TYPE "LBP_typeHMI"
TITLE = Operator panel signals / Signaux pupitre opérateur
// User data type for block LBP_HMI [DB19] / Type de données utilisateur pour bloc LBP_HMI [DB19]
   STRUCT
      A_SCLight : Bool;   // Screen light / Éclaircir écran
      A_SCDark : Bool;   // Screen darkening / Obscurcissement écran
      A_KeyDisable : Bool;   // Key disable / Désactiver touche
      A_ClearCanAl : Bool;   // Clear cancel alarms / Supprimer alarmes d'abandon
      A_ClearRecAl : Bool;   // Clear recall alarms / Supprimer alarmes de rappel
      f0_5 : Bool;
      A_SafeActionLog : Bool;   // Edge change 0 → 1: Save ACTION.COM to CRASH.COM / Front 0 → 1 : enregistrer ACTION.COM dans CRASH.COM
      A_ActWCS : Bool;   // Actual value in WCS 0=MCS / Valeur réelle dans WCS 0=MCS
      A_PLCExtViewerReject : Bool;   // External viewer reject / Refuser visualiseur externe
      A_PLCExtViewerMode : Bool;   // External viewer mode / Mode visualiseur externe
      f1_2 : Bool;
      f1_3 : Bool;
      f1_4 : Bool;
      f1_5 : Bool;
      f1_6 : Bool;
      f1_7 : Bool;
      A_1stError1 : Word;   // 1st error HIGRAPH / 1re erreur HIGRAPH
      A_1stError2 : Word;   // 1st error HIGRAPH / 1re erreur HIGRAPH
      A_ASpi1percent : Byte;   // Analog spindle 1: / Broche analogique 1 :
      A_ASpi2percent : Byte;
      A_MCPChan : Byte;
      A_OEM1 : Bool;
      A_OEM2 : Bool;
      A_AToolMeas : Bool;   // AutoToolMeasure
      f9_3 : Bool;
      f9_4 : Bool;
      f9_5 : Bool;
      f9_6 : Bool;
      f9_7 : Bool;
      A_Hardkey : Byte;   // PLC hardkeys / Touches matérielles AP
      f11 : Byte;   // Reserved for hardkeys / Réservé pour touches matérielles
      f12_0 : Bool;
      f12_1 : Bool;
      A_COM2 : Bool;
      A_COM1 : Bool;
      A_V24stop : Bool;
      A_V24ext : Bool;
      A_V24off : Bool;
      A_V24on : Bool;
      A_TeachDisable : Bool;
      f13_1 : Bool;
      f13_2 : Bool;
      f13_3 : Bool;
      f13_4 : Bool;
      A_PPdeload : Bool;
      A_PPload : Bool;
      A_PPsel : Bool;
      A_V24Index1 : Byte;
      A_V24Index2 : Byte;
      A_V24NoFile1 : Byte;
      A_V24NoFile2 : Byte;
      A_res18 : Byte;
      A_res19 : Byte;   // Message counter / Compteur de messages
      f20_0 : Bool;
      E_SCDark : Bool;   // Screen darkening / Obscurcissement écran
      E_Cancel : Bool;   // Cancel / Abandon
      E_CanCleared : Bool;   // Cancel alarms cleared / Alarmes d'abandon supprimées
      E_RecCleared : Bool;   // Recall alarms cleared / Alarmes de rappel supprimées
      f20_5 : Bool;   // res. language / rés. langue
      E_SimActiv : Bool;   // Simulation active
      E_ActWCS : Bool;   // Switchover MCS/WCS 0=MCS / Commutation MCS/WCS 0=MCS
      E_ActivWA : Byte;
      E_Chan : Byte;   // Channel displayed / Canal affiché
      E_KeybHandl : Bool;   // Keyboard handling / Gestion clavier
      E_DataTransf : Bool;   // Data transfer active / Transmission de données active
      E_DisplChange : Bool;   // Display change / Modification affichage
      f23_3 : Bool;
      f23_4 : Bool;
      f23_5 : Bool;
      f23_6 : Bool;
      f23_7 : Bool;
      E_ScreenNo : Word;
      E_res26_0 : Bool;   // Reserved / Réservé
      E_PPOK : Bool;   // Part program status OK / État programme pièce OK
      E_PPErr : Bool;   // Part program status error / Programme pièce erreur d'état
      E_PPAct : Bool;   // Part program status active / État programme pièce actif
      f26_4 : Bool;   // Reserved / Réservé
      E_PPdeload : Bool;   // Part program status deloading / État programme pièce en cours de déchargement
      E_PPload : Bool;   // Part program status loading / État programme pièce en cours de chargement
      E_PPsel : Bool;   // Part program status selecting / État programme pièce en cours de sélection
      E_PPError : Byte;   // Part program status error / Programme pièce erreur d'état
      A_PictNo : Int;
      A_PictOn : Bool;
      A_PictOff : Bool;
      f30_2 : Bool;
      f30_3 : Bool;
      f30_4 : Bool;
      f30_5 : Bool;
      f30_6 : Bool;
      f30_7 : Bool;
      E_PictOK : Bool;
      E_PictOn : Bool;
      E_PictAct : Bool;
      E_PictOff : Bool;
      E_PictErr : Bool;
      f31_5 : Bool;
      f31_6 : Bool;
      E_NotAct : Bool;
      A_FuncNo : Byte;
      A_Par1 : Byte;
      A_Par2 : Byte;
      A_Par3 : Byte;
      E_FuncErr : Byte;
      f37 : Byte;
      f38 : Byte;
      f39 : Byte;
      res40 : Array[0..9] of Byte;
      MMC2 : Struct
         A_SCLight : Bool;   // Screen light / Éclaircir écran
         A_SCDark : Bool;   // Screen darkening / Obscurcissement écran
         A_KeyDisable : Bool;   // Key disable / Désactiver touche
         A_ClearCanAl : Bool;   // Clear cancel alarms / Supprimer alarmes d'abandon
         A_ClearRecAl : Bool;   // Clear recall alarms / Supprimer alarmes de rappel
         f0_5 : Bool;
         f0_6 : Bool;
         A_ActWCS : Bool;   // Actual value in WCS 0=MCS / Valeur réelle dans WCS 0=MCS
         A_PLCExtViewerReject : Bool;   // External viewer reject / Refuser visualiseur externe
         A_PLCExtViewerMode : Bool;   // External viewer mode / Mode visualiseur externe
         f1_2 : Bool;
         f1_3 : Bool;
         f1_4 : Bool;
         f1_5 : Bool;
         f1_6 : Bool;
         f1_7 : Bool;
         A_1stError1 : Word;   // 1st error HIGRAPH / 1re erreur HIGRAPH
         A_1stError2 : Word;   // 1st error HIGRAPH / 1re erreur HIGRAPH
         A_ASpi1percent : Byte;   // Analog spindle 1: / Broche analogique 1 :
         A_ASpi2percent : Byte;
         A_MCPChan : Byte;
         A_OEM1 : Bool;
         A_OEM2 : Bool;
         A_AToolMeas : Bool;   // AutoToolMeasure
         f9_3 : Bool;
         f9_4 : Bool;
         f9_5 : Bool;
         f9_6 : Bool;
         f9_7 : Bool;
         A_Hardkey : Byte;   // PLC hardkeys / Touches matérielles AP
         f11 : Byte;   // Reserved for hardkeys / Réservé pour touches matérielles
         f12_0 : Bool;
         f12_1 : Bool;
         A_COM2 : Bool;
         A_COM1 : Bool;
         A_V24stop : Bool;
         A_V24ext : Bool;
         A_V24off : Bool;
         A_V24on : Bool;
         A_TeachDisable : Bool;
         f13_1 : Bool;
         f13_2 : Bool;
         f13_3 : Bool;
         f13_4 : Bool;
         A_PPdeload : Bool;
         A_PPload : Bool;
         A_PPsel : Bool;
         A_V24Index1 : Byte;
         A_V24Index2 : Byte;
         A_V24NoFile1 : Byte;
         A_V24NoFile2 : Byte;
         A_res18 : Byte;
         A_res19 : Byte;   // Message counter / Compteur de messages
         f20_0 : Bool;
         E_SCDark : Bool;   // Screen darkening / Obscurcissement écran
         E_Cancel : Bool;   // Cancel / Abandon
         E_CanCleared : Bool;   // Cancel alarms cleared / Alarmes d'abandon supprimées
         E_RecCleared : Bool;   // Recall alarms cleared / Alarmes de rappel supprimées
         f20_5 : Bool;   // res. language / rés. langue
         E_SimActiv : Bool;   // Simulation active
         E_ActWCS : Bool;   // Switchover MCS/WCS 0=MCS / Commutation MCS/WCS 0=MCS
         E_ActivWA : Byte;
         E_Chan : Byte;   // Channel displayed / Canal affiché
         E_KeybHandl : Bool;   // Keyboard handling / Gestion clavier
         E_DataTransf : Bool;   // Data transfer active / Transmission de données active
         E_DisplChange : Bool;   // Display change / Modification affichage
         f23_3 : Bool;
         f23_4 : Bool;
         f23_5 : Bool;
         f23_6 : Bool;
         f23_7 : Bool;
         E_ScreenNo : Word;
         E_res26_0 : Bool;   // Reserved / Réservé
         E_PPOK : Bool;   // Part program status OK / État programme pièce OK
         E_PPErr : Bool;   // Part program status error / Programme pièce erreur d'état
         E_PPAct : Bool;   // Part program status active / État programme pièce actif
         f26_4 : Bool;   // Reserved / Réservé
         E_PPdeload : Bool;   // Part program status deloading / État programme pièce en cours de déchargement
         E_PPload : Bool;   // Part program status loading / État programme pièce en cours de chargement
         E_PPsel : Bool;   // Part program status selecting / État programme pièce en cours de sélection
         E_PPError : Byte;   // Part program status error / Programme pièce erreur d'état
         A_PictNo : Int;
         A_PictOn : Bool;
         A_PictOff : Bool;
         f30_2 : Bool;
         f30_3 : Bool;
         f30_4 : Bool;
         f30_5 : Bool;
         f30_6 : Bool;
         f30_7 : Bool;
         E_PictOK : Bool;
         E_PictOn : Bool;
         E_PictAct : Bool;
         E_PictOff : Bool;
         E_PictErr : Bool;
         f31_5 : Bool;
         f31_6 : Bool;
         E_NotAct : Bool;
         A_FuncNo : Byte;
         A_Par1 : Byte;
         A_Par2 : Byte;
         A_Par3 : Byte;
         E_FuncErr : Byte;
         f37 : Byte;
         f38 : Byte;
         f39 : Byte;
         res40 : Array[0..9] of Byte;
      END_STRUCT;
      ONL_REQUEST : Word;
      ONL_CONFIRM : Word;
      PAR_CLIENT_IDENT : Word;
      PAR_MMC_TYP : Byte;
      PAR_MSTT_ADR : Byte;
      PAR_STATUS : Byte;
      PAR_Z_INFO : Byte;
      MtoNAlive : Word;
      f112 : Byte;
      ParOpKeyAdr : Byte;
      ParTcuIndex : Byte;
      f115 : Byte;
      Tcu1KeyAdr : Byte;
      Tcu2KeyAdr : Byte;
      Tcu1Index : Byte;
      Tcu2Index : Byte;
      MMC1_CLIENT_IDENT : Word;
      MMC1_TYP : Byte;
      MMC1_MSTT_ADR : Byte;
      MMC1_STATUS : Byte;
      MMC1_Z_INFO : Byte;
      MMC1_SHIFT_LOCK : Bool;
      MMC1_MSTT_SHIFT_LOCK : Bool;
      MMC1_ACTIVE_REQ : Bool;
      MMC1_ACTIVE_PERM : Bool;
      MMC1_ACTIVE_CHANGED : Bool;
      MMC1_CHANGED_DENIED : Bool;
      MMC1_TCU_SHIFT_LOCK : Bool;
      f127 : Byte;
      MMC1_TRANS_DB : Word;
      MMC2_CLIENT_IDENT : Word;
      MMC2_TYP : Byte;
      MMC2_MSTT_ADR : Byte;
      MMC2_STATUS : Byte;
      MMC2_Z_INFO : Byte;
      MMC2_SHIFT_LOCK : Bool;
      MMC2_MSTT_SHIFT_LOCK : Bool;
      MMC2_ACTIVE_REQ : Bool;
      MMC2_ACTIVE_PERM : Bool;
      MMC2_ACTIVE_CHANGED : Bool;
      MMC2_CHANGED_DENIED : Bool;
      MMC2_TCU_SHIFT_LOCK : Bool;
      f137 : Byte;
      MMC2_TRANS_DB : Word;
      A_Subtype : Int;   // For code carrier Input from PLC / Pour porte-code entrée par AP
      A_Duplo : Int;
      A_Ident : String[32];
      A_Tnumber : Int;
      A_MagazinePlace : Int;
      A_MagazinePlaceType : Int;
      A_ToolSize_Upper : Byte;
      A_ToolSize_Down : Byte;
      A_ToolSize_Left : Byte;
      A_ToolSize_Right : Byte;
      A_Channel : Byte;
      A_LoadingPlace : Byte;
      A_Magazine : Int;
      A_Unit : Byte;
      A_NCU_Index : Byte;
      A_FileIndex : Int;
      A_ActiveEnable : Bool;
      A_Override : Bool;
      A_LoadTool : Bool;
      A_DeleteTool : Bool;
      E_Subtype : Int;   // For code carrier Output to PLC / Pour porte-code sortie vers AP
      E_Duplo : Int;
      E_Ident : String[32];
      E_Tnumber : Int;
      E_ToolState : Int;
      E_MagazinePlaceType : Int;
      E_ToolSize_Upper : Byte;
      E_ToolSize_Down : Byte;
      E_ToolSize_Left : Byte;
      E_ToolSize_Right : Byte;
      E_Magazine : Int;
      E_MagazinePlace : Int;
      A_ReqMMC1 : Bool;   // For code carrier Request MMC-Interface1 / Pour porte-code demander interface MMC1
      A_ReqMMC2 : Bool;   // For code carrier Request MMC-Interface2 / Pour porte-code demander interface MMC2
      A_K_Code : Byte;
      E_Done : Bool;
      E_Error : Bool;
      E_Active : Bool;
      f252_3 : Bool;
      f252_4 : Bool;
      f252_5 : Bool;
      f252_6 : Bool;
      E_Ident_Ready : Bool;
      E_K_CodeError : Byte;   // Identify for Error_Code / Identifier pour Error_Code
      E_Error_Code : Int;
      E_Req : Bool;   // For Positioning / Pour positionnement
      f257 : Byte;
      A_Done : Bool;
      A_Error : Bool;
      A_Active : Bool;
      f258_3 : Bool;
      f258_4 : Bool;
      f258_5 : Bool;
      f258_6 : Bool;
      f258_7 : Bool;
      E_TDC_Read : Bool;
      E_TDC_Write : Bool;
      E_TDC_Cancel : Bool;
      E_TDC_Read_before_Write : Bool;
      f259_4 : Bool;
      f259_5 : Bool;
      f259_6 : Bool;
      f259_7 : Bool;
      A_Error_Code : Int;
      E_PMagazine : Int;
      E_PMagazinePlace : Int;
      E_PTnumber : Int;   // TPM data / Données TPM
      A_TPMStatus : Int;
      A_TPMCounter : Array[1..32] of DInt;
      A_HWeelSimOvr : Byte;
      f399 : Byte;
      A_SimOvr : Int;   // Simulation override / Correction simulation
      A_SimState : Int;   // Simulation state / État simulation
      E_HmiUserKey : Array[1..64] of Bool;   // HMI user keys for HMI sidescreen / HMI touches utilisateur pour écran latéral IHM
      A_HmiUserLed : Array[1..64] of Bool;   // LEDs to the user keys for HMI sidescreen / LED pour touches utilisateur pour écran latéral IHM
      A_DisableHmiUserKey : Array[1..64] of Bool;   // Disable user keys for HMI sidescreen / Désactiver les touches utilisateur pour écran latéral IHM
      SafetyAutoAcceptanceTest : Struct   // Interface for the automated acceptance test
         E_Prepare : Bool;   // Prepare automated acceptance test requested by client
         E_Finalize : Bool;   // Stop automated acceptance test requested by client
         E_Cancel : Bool;   // Cancel automated acceptance test requested by client
         E_Perform : Bool;   // Perform automated acceptance test requested by client
         E_PerformSequence : Bool;   // Perform entire test sequence for automated acceptance test requested by client
         f428_5 : Bool;
         f428_6 : Bool;
         f428_7 : Bool;
         f429 : Byte;
         A_Prepared : Bool;   // Automated acceptance test was successfully prepared
         A_Finalized : Bool;   // Automated acceptance test was successfully stopped
         A_Canceled : Bool;   // Automated acceptance test was canceled successfully
         A_Performed : Bool;   // Automated acceptance test was performed successfully
         A_SequencePerformed : Bool;   // Entire test sequence for automated acceptance test is running
         f430_5 : Bool;
         f430_6 : Bool;
         f430_7 : Bool;
         f431_0 : Bool;
         A_Error : Bool;   // Automated acceptance test was canceled
         A_InvalidGroup : Bool;   // Test group is not accepted
         A_InvalidNumber : Bool;   // Test number is not accepted
         f431_4 : Bool;
         f431_5 : Bool;
         f431_6 : Bool;
         f431_7 : Bool;
         E_Group : Int;   // Test group for the current test
         E_Number : Int;   // Test number for the current test
         E_AxisNumber : Int;   // Axis number for the current test
         E_TraversePlus : Bool;   // Traversing direction for the current test (FALSE=negative, TRUE=positive)
         E_SelectSafeStop : Bool;   // Safe Stop is set for the current test
         E_SelectBrake : Bool;   // Brake used for the current test. (FALSE=Brake1, TRUE=Brake2)
         E_SelectSbtMode : Bool;   // SBT Test Sequence used for the current test. (FALSE=Sequence1, TRUE=Sequence2)
         E_SelectSlpMode : Int;   // Safe End Position used for the current test. ("SE/SLP PositionArea" : 1=SE1 ; 2=SE2)
         E_SelectSlsMode : Int;   // Safe Speed (SG1..SG4) used for the current test
      END_STRUCT;
   END_STRUCT;
END_TYPE

TYPE "LBP_typeInternal1"
TITLE = Internal data type for basic program / Type de données interne pour programme de base
// Data type only for internal use in the basic program / Type de données réservé à l'utilisation interne dans le programme de base
   STRUCT
      active : Bool;
      mcpAddress : USInt;
      modeDCK : Bool;
      clientPort : UInt;
      connectionId : CONN_OUC;
      mcpClientReference : Word;
      mcpInPointer : Struct
         DbNumber : Word;
         PointerAddress : DWord;
      END_STRUCT;
      mcpOutPointer : Struct
         DbNumber : Word;
         PointerAddress : DWord;
      END_STRUCT;
      mcpDefaultInLength : UInt;
      mcpDefaultOutLength : UInt;
      useIpAddress : Bool;
      ipAddress : Array[1..4] of USInt;
   END_STRUCT;
END_TYPE

TYPE "LBP_typeInternal2"
TITLE = Internal data type for basic program / Type de données interne pour programme de base
// Data type only for internal use in the basic program / Type de données réservé à l'utilisation interne dans le programme de base
   STRUCT
      "Version" { ExternalAccessible := 'False'; ExternalVisible := 'False'; ExternalWritable := 'False'} : UDInt;
      ObNumber { ExternalAccessible := 'False'; ExternalVisible := 'False'; ExternalWritable := 'False'} : UDInt;
   END_STRUCT;
END_TYPE

TYPE "LBP_typeInternal3"
TITLE = Internal data type for basic program / Type de données interne pour programme de base
// Data type only for internal use in the basic program / Type de données réservé à l'utilisation interne dans le programme de base
   STRUCT
      "Version" { ExternalAccessible := 'False'; ExternalVisible := 'False'; ExternalWritable := 'False'} : UDInt;
      BlockReturnValue { ExternalAccessible := 'False'; ExternalVisible := 'False'; ExternalWritable := 'False'} : UDInt;
      AlarmList { ExternalAccessible := 'False'; ExternalVisible := 'False'; ExternalWritable := 'False'} : Array[1..6] of Struct
         ARID : UInt;
         AlarmMessage : Bool;
         OperationMessage : Bool;
         AlarmIsComing : Bool;
         StopPlc : Bool;
         NumberOfExtendedValues : USInt;
         AlarmNumber : UDInt;
         ExtendedValueList : Array[1..9] of UDInt;
      END_STRUCT;
   END_STRUCT;
END_TYPE

TYPE "LBP_typeInternal4"
TITLE = Internal data type for basic program / Type de données interne pour programme de base
// Data type only for internal use in the basic program / Type de données réservé à l'utilisation interne dans le programme de base
   STRUCT
      Handwheels : Array[1..6] of Struct
         active : Bool;
         recent : Bool;
         stopped : Bool;
         pulses : Int;
      END_STRUCT;
   END_STRUCT;
END_TYPE

TYPE "LBP_typeInternal5"
TITLE = Internal data type for basic program / Type de données interne pour programme de base
// Data type only for internal use in the basic program / Type de données réservé à l'utilisation interne dans le programme de base
   STRUCT
      accepted : Bool;
      abort : Bool;
      writeRecord : Bool;
      mcpNumber : UInt;
      slotNumber : UInt;
      recordNumber : UInt;
      recordLength : UInt;
      recordData : Array[0..223] of Byte;
      done : Bool;
      busy : Bool;
      error : Bool;
      status : Word;
   END_STRUCT;
END_TYPE

TYPE "LBP_typeModeGroup"
TITLE = Mode group signals / Signaux groupe de modes de fonctionnement
// User data type for block LBP_ModeGroup [DB11] / Type de données utilisateur pour bloc LBP_ModeGroup [DB11]
   STRUCT
      A_AUTO : Bool;   // Operating mode AUTOMATIC / Mode AUTOMATIC
      A_MDA : Bool;   // Operating mode MDA / Mode MDA
      A_JOG : Bool;   // Operating mode JOG / Mode JOG
      f0_3 : Bool;
      A_MCDisable : Bool;   // Mode change disable / Désactiver changement mode de fonctionnement
      A_MGStop : Bool;   // Mode group stop / Groupe de modes de fonctionnement Arrêt
      A_MGStopASp : Bool;   // Mode group stop axes plus spindle / Groupe de modes de fonctionnement Arrêt axes et broche
      A_MGReset : Bool;   // Mode group reset / Groupe de modes de fonctionnement Reset
      A_TEACHIN : Bool;   // Machine function TEACH IN / Fonction machine TEACH IN
      A_REPOS : Bool;   // Machine function REPOS / Fonction machine REPOS
      A_REF : Bool;   // Machine function REF / Fonction machine REF
      f1_3 : Bool;
      f1_4 : Bool;
      f1_5 : Bool;
      A_SingleBlock_B : Bool;   // Single block type B / Bloc par bloc type B
      A_SingleBlock_A : Bool;   // Single block type A / Bloc par bloc type A
      A_INC1 : Bool;   // INC1
      A_INC10 : Bool;   // INC10
      A_INC100 : Bool;   // INC100
      A_INC1000 : Bool;   // INC1000
      A_INC10000 : Bool;   // INC10000
      A_INCVar : Bool;   // INC variable / Variable INC
      A_ContManTravel : Bool;   // Continuous manual travel / Mode manuel continu
      f2_7 : Bool;
      f3 : Byte;
      E_MMC_AUTO : Bool;   // HMI mode strobe AUTOMATIC / HMI mode Strobe AUTOMATIC
      E_MMC_MDA : Bool;   // HMI mode strobe MDA / HMI mode Strobe MDA
      E_MMC_JOG : Bool;   // HMI mode strobe JOG / HMI mode Strobe JOG
      f4_3 : Bool;
      f4_4 : Bool;
      f4_5 : Bool;
      f4_6 : Bool;
      f4_7 : Bool;
      E_MMC_TEACHIN : Bool;   // HMI machine function strobe TEACH IN / HMI Fonction machine Strobe TEACH IN
      E_MMC_REPOS : Bool;   // HMI machine function strobe REPOS / HMI Fonction machine Strobe REPOS
      E_MMC_REF : Bool;   // HMI machine function strobe REF / HMI Fonction machine Strobe REF
      f5_3 : Bool;
      f5_4 : Bool;
      f5_5 : Bool;
      f5_6 : Bool;
      f5_7 : Bool;
      E_AUTO : Bool;   // Active operating mode AUTOMATIC / Mode actif AUTOMATIC
      E_MDA : Bool;   // Active operating mode MDA / Mode actif MDA
      E_JOG : Bool;   // Active operating mode JOG / Mode actif JOG
      E_MGOK : Bool;   // Mode group ready / Groupe de modes de fonctionnement prêt
      E_MGreseted : Bool;   // Mode group reset performed / Groupe de modes de fonctionnement Reset effectué
      E_NCKintJOG : Bool;   // NCK internal JOG active / NCK JOG interne actif
      f6_6 : Bool;
      E_ChanReset : Bool;   // All channels in reset state / Tous les canaux en mode Reset
      E_TEACHIN : Bool;   // Active machine function TEACH IN / Fonction machine active TEACH IN
      E_REPOS : Bool;   // Active machine function REPOS / Fonction machine active REPOS
      E_REF : Bool;   // Active machine function REF / Fonction machine active REF
      f7_3 : Bool;
      f7_4 : Bool;
      f7_5 : Bool;
      f7_6 : Bool;
      f7_7 : Bool;
      E_INC1 : Bool;   // INC1
      E_INC10 : Bool;   // INC10
      E_INC100 : Bool;   // INC100
      E_INC1000 : Bool;   // INC1000
      E_INC10000 : Bool;   // INC10000
      E_INCVar : Bool;   // INC variable / Variable INC
      E_ContManTravelAct : Bool;   // Continuous manual travel active / Mode manuel continu actif
      f8_7 : Bool;
      f9 : Byte;
      E_HMI_INC1 : Bool;   // INC1 from HMI / INC1 depuis IHM
      E_HMI_INC10 : Bool;   // INC10 from HMI / INC10 depuis IHM
      E_HMI_INC100 : Bool;   // INC100 from HMI / INC100 depuis IHM
      E_HMI_INC1000 : Bool;   // INC1000 from HMI / INC1000 depuis IHM
      E_HMI_INC10000 : Bool;   // INC10000 from HMI / INC10000 depuis IHM
      E_HMI_INCVar : Bool;   // INC variable from HMI / Variable INC depuis IHM
      E_HMI_ContManTravel : Bool;   // Continuous manual travel active from HMI / Course manuelle continue active depuis IHM
      f10_7 : Bool;
      f11 : Byte;
      f12 : Array[12..19] of Byte;
      MG : Array[2..10] of Struct   // next mode group from DBB20, as before / groupe de mode suivant depuis DBB20, comme avant
         A_AUTO : Bool;   // Operating mode AUTOMATIC / Mode AUTOMATIC
         A_MDA : Bool;   // Operating mode MDA / Mode MDA
         A_JOG : Bool;   // Operating mode JOG / Mode JOG
         f0_3 : Bool;
         A_MCDisable : Bool;   // Mode change disable / Désactiver changement mode de fonctionnement
         A_MGStop : Bool;   // Mode group stop / Groupe de modes de fonctionnement Arrêt
         A_MGStopASp : Bool;   // Mode group stop axes plus spindle / Groupe de modes de fonctionnement Arrêt axes et broche
         A_MGReset : Bool;   // Mode group reset / Groupe de modes de fonctionnement Reset
         A_TEACHIN : Bool;   // Machine function TEACH IN / Fonction machine TEACH IN
         A_REPOS : Bool;   // Machine function REPOS / Fonction machine REPOS
         A_REF : Bool;   // Machine function REF / Fonction machine REF
         f1_3 : Bool;
         f1_4 : Bool;
         f1_5 : Bool;
         A_SingleBlock_B : Bool;   // Single block type B / Bloc par bloc type B
         A_SingleBlock_A : Bool;   // Single block type A / Bloc par bloc type A
         A_INC1 : Bool;   // INC1
         A_INC10 : Bool;   // INC10
         A_INC100 : Bool;   // INC100
         A_INC1000 : Bool;   // INC1000
         A_INC10000 : Bool;   // INC10000
         A_INCVar : Bool;   // INC variable / Variable INC
         A_ContManTravel : Bool;   // Continuous manual travel / Mode manuel continu
         f2_7 : Bool;
         f3 : Byte;
         E_MMC_AUTO : Bool;   // HMI mode strobe AUTOMATIC / HMI mode Strobe AUTOMATIC
         E_MMC_MDA : Bool;   // HMI mode strobe MDA / HMI mode Strobe MDA
         E_MMC_JOG : Bool;   // HMI mode strobe JOG / HMI mode Strobe JOG
         f4_3 : Bool;
         f4_4 : Bool;
         f4_5 : Bool;
         f4_6 : Bool;
         f4_7 : Bool;
         E_MMC_TEACHIN : Bool;   // HMI machine function strobe TEACH IN / HMI Fonction machine Strobe TEACH IN
         E_MMC_REPOS : Bool;   // HMI machine function strobe REPOS / HMI Fonction machine Strobe REPOS
         E_MMC_REF : Bool;   // HMI machine function strobe REF / HMI Fonction machine Strobe REF
         f5_3 : Bool;
         f5_4 : Bool;
         f5_5 : Bool;
         f5_6 : Bool;
         f5_7 : Bool;
         E_AUTO : Bool;   // Active operating mode AUTOMATIC / Mode actif AUTOMATIC
         E_MDA : Bool;   // Active operating mode MDA / Mode actif MDA
         E_JOG : Bool;   // Active operating mode JOG / Mode actif JOG
         E_MGOK : Bool;   // Mode group ready / Groupe de modes de fonctionnement prêt
         E_MGreseted : Bool;   // Mode group reset / Groupe de modes de fonctionnement Reset
         E_NCKintJOG : Bool;   // NCK internal JOG active / NCK JOG interne actif
         f6_6 : Bool;
         E_ChanReset : Bool;   // All channels in reset state / Tous les canaux en mode Reset
         E_TEACHIN : Bool;   // Active machine function TEACH IN / Fonction machine active TEACH IN
         E_REPOS : Bool;   // Active machine function REPOS / Fonction machine active REPOS
         E_REF : Bool;   // Active machine function REF / Fonction machine active REF
         f7_3 : Bool;
         f7_4 : Bool;
         f7_5 : Bool;
         f7_6 : Bool;
         f7_7 : Bool;
         E_INC1 : Bool;   // INC1
         E_INC10 : Bool;   // INC10
         E_INC100 : Bool;   // INC100
         E_INC1000 : Bool;   // INC1000
         E_INC10000 : Bool;   // INC10000
         E_INCVar : Bool;   // INC variable / Variable INC
         E_ContManTravelAct : Bool;   // Continuous manual travel active / Mode manuel continu actif
         f8_7 : Bool;
         f9 : Byte;
         E_HMI_INC1 : Bool;   // INC1 from HMI / INC1 depuis IHM
         E_HMI_INC10 : Bool;   // INC10 from HMI / INC10 depuis IHM
         E_HMI_INC100 : Bool;   // INC100 from HMI / INC100 depuis IHM
         E_HMI_INC1000 : Bool;   // INC1000 from HMI / INC1000 depuis IHM
         E_HMI_INC10000 : Bool;   // INC10000 from HMI / INC10000 depuis IHM
         E_HMI_INCVar : Bool;   // INC variable from HMI / Variable INC depuis IHM
         E_HMI_ContManTravel : Bool;   // Continuous manual travel active from HMI / Course manuelle continue active depuis IHM
         f10_7 : Bool;
         f11 : Byte;
         f12 : Array[12..19] of Byte;
      END_STRUCT;
   END_STRUCT;
   // // MG[3].A_AUTO : Operating mode AUTOMATIC / Mode AUTOMATIC
   // // MG[4].A_AUTO : Operating mode AUTOMATIC / Mode AUTOMATIC
   // // MG[5].A_AUTO : Operating mode AUTOMATIC / Mode AUTOMATIC
   // // MG[6].A_AUTO : Operating mode AUTOMATIC / Mode AUTOMATIC
   // // MG[7].A_AUTO : Operating mode AUTOMATIC / Mode AUTOMATIC
   // // MG[8].A_AUTO : Operating mode AUTOMATIC / Mode AUTOMATIC
   // // MG[9].A_AUTO : Operating mode AUTOMATIC / Mode AUTOMATIC
   // // MG[10].A_AUTO : Operating mode AUTOMATIC / Mode AUTOMATIC
   // // MG[3].A_MDA : Operating mode MDA / Mode MDA
   // // MG[4].A_MDA : Operating mode MDA / Mode MDA
   // // MG[5].A_MDA : Operating mode MDA / Mode MDA
   // // MG[6].A_MDA : Operating mode MDA / Mode MDA
   // // MG[7].A_MDA : Operating mode MDA / Mode MDA
   // // MG[8].A_MDA : Operating mode MDA / Mode MDA
   // // MG[9].A_MDA : Operating mode MDA / Mode MDA
   // // MG[10].A_MDA : Operating mode MDA / Mode MDA
   // // MG[3].A_JOG : Operating mode JOG / Mode JOG
   // // MG[4].A_JOG : Operating mode JOG / Mode JOG
   // // MG[5].A_JOG : Operating mode JOG / Mode JOG
   // // MG[6].A_JOG : Operating mode JOG / Mode JOG
   // // MG[7].A_JOG : Operating mode JOG / Mode JOG
   // // MG[8].A_JOG : Operating mode JOG / Mode JOG
   // // MG[9].A_JOG : Operating mode JOG / Mode JOG
   // // MG[10].A_JOG : Operating mode JOG / Mode JOG
   // // MG[3].A_MCDisable : Mode change disable / Désactiver changement mode de fonctionnement
   // // MG[4].A_MCDisable : Mode change disable / Désactiver changement mode de fonctionnement
   // // MG[5].A_MCDisable : Mode change disable / Désactiver changement mode de fonctionnement
   // // MG[6].A_MCDisable : Mode change disable / Désactiver changement mode de fonctionnement
   // // MG[7].A_MCDisable : Mode change disable / Désactiver changement mode de fonctionnement
   // // MG[8].A_MCDisable : Mode change disable / Désactiver changement mode de fonctionnement
   // // MG[9].A_MCDisable : Mode change disable / Désactiver changement mode de fonctionnement
   // // MG[10].A_MCDisable : Mode change disable / Désactiver changement mode de fonctionnement
   // // MG[3].A_MGStop : Mode group stop / Groupe de modes de fonctionnement Arrêt
   // // MG[4].A_MGStop : Mode group stop / Groupe de modes de fonctionnement Arrêt
   // // MG[5].A_MGStop : Mode group stop / Groupe de modes de fonctionnement Arrêt
   // // MG[6].A_MGStop : Mode group stop / Groupe de modes de fonctionnement Arrêt
   // // MG[7].A_MGStop : Mode group stop / Groupe de modes de fonctionnement Arrêt
   // // MG[8].A_MGStop : Mode group stop / Groupe de modes de fonctionnement Arrêt
   // // MG[9].A_MGStop : Mode group stop / Groupe de modes de fonctionnement Arrêt
   // // MG[10].A_MGStop : Mode group stop / Groupe de modes de fonctionnement Arrêt
   // // MG[3].A_MGStopASp : Mode group stop axes plus spindle / Groupe de modes de fonctionnement Arrêt axes et broche
   // // MG[4].A_MGStopASp : Mode group stop axes plus spindle / Groupe de modes de fonctionnement Arrêt axes et broche
   // // MG[5].A_MGStopASp : Mode group stop axes plus spindle / Groupe de modes de fonctionnement Arrêt axes et broche
   // // MG[6].A_MGStopASp : Mode group stop axes plus spindle / Groupe de modes de fonctionnement Arrêt axes et broche
   // // MG[7].A_MGStopASp : Mode group stop axes plus spindle / Groupe de modes de fonctionnement Arrêt axes et broche
   // // MG[8].A_MGStopASp : Mode group stop axes plus spindle / Groupe de modes de fonctionnement Arrêt axes et broche
   // // MG[9].A_MGStopASp : Mode group stop axes plus spindle / Groupe de modes de fonctionnement Arrêt axes et broche
   // // MG[10].A_MGStopASp : Mode group stop axes plus spindle / Groupe de modes de fonctionnement Arrêt axes et broche
   // // MG[3].A_MGReset : Mode group reset / Groupe de modes de fonctionnement Reset
   // // MG[4].A_MGReset : Mode group reset / Groupe de modes de fonctionnement Reset
   // // MG[5].A_MGReset : Mode group reset / Groupe de modes de fonctionnement Reset
   // // MG[6].A_MGReset : Mode group reset / Groupe de modes de fonctionnement Reset
   // // MG[7].A_MGReset : Mode group reset / Groupe de modes de fonctionnement Reset
   // // MG[8].A_MGReset : Mode group reset / Groupe de modes de fonctionnement Reset
   // // MG[9].A_MGReset : Mode group reset / Groupe de modes de fonctionnement Reset
   // // MG[10].A_MGReset : Mode group reset / Groupe de modes de fonctionnement Reset
   // // MG[3].A_TEACHIN : Machine function TEACH IN / Fonction machine TEACH IN
   // // MG[4].A_TEACHIN : Machine function TEACH IN / Fonction machine TEACH IN
   // // MG[5].A_TEACHIN : Machine function TEACH IN / Fonction machine TEACH IN
   // // MG[6].A_TEACHIN : Machine function TEACH IN / Fonction machine TEACH IN
   // // MG[7].A_TEACHIN : Machine function TEACH IN / Fonction machine TEACH IN
   // // MG[8].A_TEACHIN : Machine function TEACH IN / Fonction machine TEACH IN
   // // MG[9].A_TEACHIN : Machine function TEACH IN / Fonction machine TEACH IN
   // // MG[10].A_TEACHIN : Machine function TEACH IN / Fonction machine TEACH IN
   // // MG[3].A_REPOS : Machine function REPOS / Fonction machine REPOS
   // // MG[4].A_REPOS : Machine function REPOS / Fonction machine REPOS
   // // MG[5].A_REPOS : Machine function REPOS / Fonction machine REPOS
   // // MG[6].A_REPOS : Machine function REPOS / Fonction machine REPOS
   // // MG[7].A_REPOS : Machine function REPOS / Fonction machine REPOS
   // // MG[8].A_REPOS : Machine function REPOS / Fonction machine REPOS
   // // MG[9].A_REPOS : Machine function REPOS / Fonction machine REPOS
   // // MG[10].A_REPOS : Machine function REPOS / Fonction machine REPOS
   // // MG[3].A_REF : Machine function REF / Fonction machine REF
   // // MG[4].A_REF : Machine function REF / Fonction machine REF
   // // MG[5].A_REF : Machine function REF / Fonction machine REF
   // // MG[6].A_REF : Machine function REF / Fonction machine REF
   // // MG[7].A_REF : Machine function REF / Fonction machine REF
   // // MG[8].A_REF : Machine function REF / Fonction machine REF
   // // MG[9].A_REF : Machine function REF / Fonction machine REF
   // // MG[10].A_REF : Machine function REF / Fonction machine REF
   // // MG[3].A_SingleBlock_B : Single block type B / Bloc par bloc type B
   // // MG[4].A_SingleBlock_B : Single block type B / Bloc par bloc type B
   // // MG[5].A_SingleBlock_B : Single block type B / Bloc par bloc type B
   // // MG[6].A_SingleBlock_B : Single block type B / Bloc par bloc type B
   // // MG[7].A_SingleBlock_B : Single block type B / Bloc par bloc type B
   // // MG[8].A_SingleBlock_B : Single block type B / Bloc par bloc type B
   // // MG[9].A_SingleBlock_B : Single block type B / Bloc par bloc type B
   // // MG[10].A_SingleBlock_B : Single block type B / Bloc par bloc type B
   // // MG[3].A_SingleBlock_A : Single block type A / Bloc par bloc type A
   // // MG[4].A_SingleBlock_A : Single block type A / Bloc par bloc type A
   // // MG[5].A_SingleBlock_A : Single block type A / Bloc par bloc type A
   // // MG[6].A_SingleBlock_A : Single block type A / Bloc par bloc type A
   // // MG[7].A_SingleBlock_A : Single block type A / Bloc par bloc type A
   // // MG[8].A_SingleBlock_A : Single block type A / Bloc par bloc type A
   // // MG[9].A_SingleBlock_A : Single block type A / Bloc par bloc type A
   // // MG[10].A_SingleBlock_A : Single block type A / Bloc par bloc type A
   // // MG[3].A_INC1 : INC1
   // // MG[4].A_INC1 : INC1
   // // MG[5].A_INC1 : INC1
   // // MG[6].A_INC1 : INC1
   // // MG[7].A_INC1 : INC1
   // // MG[8].A_INC1 : INC1
   // // MG[9].A_INC1 : INC1
   // // MG[10].A_INC1 : INC1
   // // MG[3].A_INC10 : INC10
   // // MG[4].A_INC10 : INC10
   // // MG[5].A_INC10 : INC10
   // // MG[6].A_INC10 : INC10
   // // MG[7].A_INC10 : INC10
   // // MG[8].A_INC10 : INC10
   // // MG[9].A_INC10 : INC10
   // // MG[10].A_INC10 : INC10
   // // MG[3].A_INC100 : INC100
   // // MG[4].A_INC100 : INC100
   // // MG[5].A_INC100 : INC100
   // // MG[6].A_INC100 : INC100
   // // MG[7].A_INC100 : INC100
   // // MG[8].A_INC100 : INC100
   // // MG[9].A_INC100 : INC100
   // // MG[10].A_INC100 : INC100
   // // MG[3].A_INC1000 : INC1000
   // // MG[4].A_INC1000 : INC1000
   // // MG[5].A_INC1000 : INC1000
   // // MG[6].A_INC1000 : INC1000
   // // MG[7].A_INC1000 : INC1000
   // // MG[8].A_INC1000 : INC1000
   // // MG[9].A_INC1000 : INC1000
   // // MG[10].A_INC1000 : INC1000
   // // MG[3].A_INC10000 : INC10000
   // // MG[4].A_INC10000 : INC10000
   // // MG[5].A_INC10000 : INC10000
   // // MG[6].A_INC10000 : INC10000
   // // MG[7].A_INC10000 : INC10000
   // // MG[8].A_INC10000 : INC10000
   // // MG[9].A_INC10000 : INC10000
   // // MG[10].A_INC10000 : INC10000
   // // MG[3].A_INCVar : INC variable / Variable INC
   // // MG[4].A_INCVar : INC variable / Variable INC
   // // MG[5].A_INCVar : INC variable / Variable INC
   // // MG[6].A_INCVar : INC variable / Variable INC
   // // MG[7].A_INCVar : INC variable / Variable INC
   // // MG[8].A_INCVar : INC variable / Variable INC
   // // MG[9].A_INCVar : INC variable / Variable INC
   // // MG[10].A_INCVar : INC variable / Variable INC
   // // MG[3].A_ContManTravel : Continuous manual travel / Mode manuel continu
   // // MG[4].A_ContManTravel : Continuous manual travel / Mode manuel continu
   // // MG[5].A_ContManTravel : Continuous manual travel / Mode manuel continu
   // // MG[6].A_ContManTravel : Continuous manual travel / Mode manuel continu
   // // MG[7].A_ContManTravel : Continuous manual travel / Mode manuel continu
   // // MG[8].A_ContManTravel : Continuous manual travel / Mode manuel continu
   // // MG[9].A_ContManTravel : Continuous manual travel / Mode manuel continu
   // // MG[10].A_ContManTravel : Continuous manual travel / Mode manuel continu
   // // MG[3].E_MMC_AUTO : HMI mode strobe AUTOMATIC / HMI mode Strobe AUTOMATIC
   // // MG[4].E_MMC_AUTO : HMI mode strobe AUTOMATIC / HMI mode Strobe AUTOMATIC
   // // MG[5].E_MMC_AUTO : HMI mode strobe AUTOMATIC / HMI mode Strobe AUTOMATIC
   // // MG[6].E_MMC_AUTO : HMI mode strobe AUTOMATIC / HMI mode Strobe AUTOMATIC
   // // MG[7].E_MMC_AUTO : HMI mode strobe AUTOMATIC / HMI mode Strobe AUTOMATIC
   // // MG[8].E_MMC_AUTO : HMI mode strobe AUTOMATIC / HMI mode Strobe AUTOMATIC
   // // MG[9].E_MMC_AUTO : HMI mode strobe AUTOMATIC / HMI mode Strobe AUTOMATIC
   // // MG[10].E_MMC_AUTO : HMI mode strobe AUTOMATIC / HMI mode Strobe AUTOMATIC
   // // MG[3].E_MMC_MDA : HMI mode strobe MDA / HMI mode Strobe MDA
   // // MG[4].E_MMC_MDA : HMI mode strobe MDA / HMI mode Strobe MDA
   // // MG[5].E_MMC_MDA : HMI mode strobe MDA / HMI mode Strobe MDA
   // // MG[6].E_MMC_MDA : HMI mode strobe MDA / HMI mode Strobe MDA
   // // MG[7].E_MMC_MDA : HMI mode strobe MDA / HMI mode Strobe MDA
   // // MG[8].E_MMC_MDA : HMI mode strobe MDA / HMI mode Strobe MDA
   // // MG[9].E_MMC_MDA : HMI mode strobe MDA / HMI mode Strobe MDA
   // // MG[10].E_MMC_MDA : HMI mode strobe MDA / HMI mode Strobe MDA
   // // MG[3].E_MMC_JOG : HMI mode strobe JOG / HMI mode Strobe JOG
   // // MG[4].E_MMC_JOG : HMI mode strobe JOG / HMI mode Strobe JOG
   // // MG[5].E_MMC_JOG : HMI mode strobe JOG / HMI mode Strobe JOG
   // // MG[6].E_MMC_JOG : HMI mode strobe JOG / HMI mode Strobe JOG
   // // MG[7].E_MMC_JOG : HMI mode strobe JOG / HMI mode Strobe JOG
   // // MG[8].E_MMC_JOG : HMI mode strobe JOG / HMI mode Strobe JOG
   // // MG[9].E_MMC_JOG : HMI mode strobe JOG / HMI mode Strobe JOG
   // // MG[10].E_MMC_JOG : HMI mode strobe JOG / HMI mode Strobe JOG
   // // MG[3].E_MMC_TEACHIN : HMI machine function strobe TEACH IN / HMI Fonction machine Strobe TEACH IN
   // // MG[4].E_MMC_TEACHIN : HMI machine function strobe TEACH IN / HMI Fonction machine Strobe TEACH IN
   // // MG[5].E_MMC_TEACHIN : HMI machine function strobe TEACH IN / HMI Fonction machine Strobe TEACH IN
   // // MG[6].E_MMC_TEACHIN : HMI machine function strobe TEACH IN / HMI Fonction machine Strobe TEACH IN
   // // MG[7].E_MMC_TEACHIN : HMI machine function strobe TEACH IN / HMI Fonction machine Strobe TEACH IN
   // // MG[8].E_MMC_TEACHIN : HMI machine function strobe TEACH IN / HMI Fonction machine Strobe TEACH IN
   // // MG[9].E_MMC_TEACHIN : HMI machine function strobe TEACH IN / HMI Fonction machine Strobe TEACH IN
   // // MG[10].E_MMC_TEACHIN : HMI machine function strobe TEACH IN / HMI Fonction machine Strobe TEACH IN
   // // MG[3].E_MMC_REPOS : HMI machine function strobe REPOS / HMI Fonction machine Strobe REPOS
   // // MG[4].E_MMC_REPOS : HMI machine function strobe REPOS / HMI Fonction machine Strobe REPOS
   // // MG[5].E_MMC_REPOS : HMI machine function strobe REPOS / HMI Fonction machine Strobe REPOS
   // // MG[6].E_MMC_REPOS : HMI machine function strobe REPOS / HMI Fonction machine Strobe REPOS
   // // MG[7].E_MMC_REPOS : HMI machine function strobe REPOS / HMI Fonction machine Strobe REPOS
   // // MG[8].E_MMC_REPOS : HMI machine function strobe REPOS / HMI Fonction machine Strobe REPOS
   // // MG[9].E_MMC_REPOS : HMI machine function strobe REPOS / HMI Fonction machine Strobe REPOS
   // // MG[10].E_MMC_REPOS : HMI machine function strobe REPOS / HMI Fonction machine Strobe REPOS
   // // MG[3].E_MMC_REF : HMI machine function strobe REF / HMI Fonction machine Strobe REF
   // // MG[4].E_MMC_REF : HMI machine function strobe REF / HMI Fonction machine Strobe REF
   // // MG[5].E_MMC_REF : HMI machine function strobe REF / HMI Fonction machine Strobe REF
   // // MG[6].E_MMC_REF : HMI machine function strobe REF / HMI Fonction machine Strobe REF
   // // MG[7].E_MMC_REF : HMI machine function strobe REF / HMI Fonction machine Strobe REF
   // // MG[8].E_MMC_REF : HMI machine function strobe REF / HMI Fonction machine Strobe REF
   // // MG[9].E_MMC_REF : HMI machine function strobe REF / HMI Fonction machine Strobe REF
   // // MG[10].E_MMC_REF : HMI machine function strobe REF / HMI Fonction machine Strobe REF
   // // MG[3].E_AUTO : Active operating mode AUTOMATIC / Mode actif AUTOMATIC
   // // MG[4].E_AUTO : Active operating mode AUTOMATIC / Mode actif AUTOMATIC
   // // MG[5].E_AUTO : Active operating mode AUTOMATIC / Mode actif AUTOMATIC
   // // MG[6].E_AUTO : Active operating mode AUTOMATIC / Mode actif AUTOMATIC
   // // MG[7].E_AUTO : Active operating mode AUTOMATIC / Mode actif AUTOMATIC
   // // MG[8].E_AUTO : Active operating mode AUTOMATIC / Mode actif AUTOMATIC
   // // MG[9].E_AUTO : Active operating mode AUTOMATIC / Mode actif AUTOMATIC
   // // MG[10].E_AUTO : Active operating mode AUTOMATIC / Mode actif AUTOMATIC
   // // MG[3].E_MDA : Active operating mode MDA / Mode actif MDA
   // // MG[4].E_MDA : Active operating mode MDA / Mode actif MDA
   // // MG[5].E_MDA : Active operating mode MDA / Mode actif MDA
   // // MG[6].E_MDA : Active operating mode MDA / Mode actif MDA
   // // MG[7].E_MDA : Active operating mode MDA / Mode actif MDA
   // // MG[8].E_MDA : Active operating mode MDA / Mode actif MDA
   // // MG[9].E_MDA : Active operating mode MDA / Mode actif MDA
   // // MG[10].E_MDA : Active operating mode MDA / Mode actif MDA
   // // MG[3].E_JOG : Active operating mode JOG / Mode actif JOG
   // // MG[4].E_JOG : Active operating mode JOG / Mode actif JOG
   // // MG[5].E_JOG : Active operating mode JOG / Mode actif JOG
   // // MG[6].E_JOG : Active operating mode JOG / Mode actif JOG
   // // MG[7].E_JOG : Active operating mode JOG / Mode actif JOG
   // // MG[8].E_JOG : Active operating mode JOG / Mode actif JOG
   // // MG[9].E_JOG : Active operating mode JOG / Mode actif JOG
   // // MG[10].E_JOG : Active operating mode JOG / Mode actif JOG
   // // MG[3].E_MGOK : Mode group ready / Groupe de modes de fonctionnement prêt
   // // MG[4].E_MGOK : Mode group ready / Groupe de modes de fonctionnement prêt
   // // MG[5].E_MGOK : Mode group ready / Groupe de modes de fonctionnement prêt
   // // MG[6].E_MGOK : Mode group ready / Groupe de modes de fonctionnement prêt
   // // MG[7].E_MGOK : Mode group ready / Groupe de modes de fonctionnement prêt
   // // MG[8].E_MGOK : Mode group ready / Groupe de modes de fonctionnement prêt
   // // MG[9].E_MGOK : Mode group ready / Groupe de modes de fonctionnement prêt
   // // MG[10].E_MGOK : Mode group ready / Groupe de modes de fonctionnement prêt
   // // MG[3].E_MGreseted : Mode group reset / Groupe de modes de fonctionnement Reset
   // // MG[4].E_MGreseted : Mode group reset / Groupe de modes de fonctionnement Reset
   // // MG[5].E_MGreseted : Mode group reset / Groupe de modes de fonctionnement Reset
   // // MG[6].E_MGreseted : Mode group reset / Groupe de modes de fonctionnement Reset
   // // MG[7].E_MGreseted : Mode group reset / Groupe de modes de fonctionnement Reset
   // // MG[8].E_MGreseted : Mode group reset / Groupe de modes de fonctionnement Reset
   // // MG[9].E_MGreseted : Mode group reset / Groupe de modes de fonctionnement Reset
   // // MG[10].E_MGreseted : Mode group reset / Groupe de modes de fonctionnement Reset
   // // MG[3].E_NCKintJOG : NCK internal JOG active / NCK JOG interne actif
   // // MG[4].E_NCKintJOG : NCK internal JOG active / NCK JOG interne actif
   // // MG[5].E_NCKintJOG : NCK internal JOG active / NCK JOG interne actif
   // // MG[6].E_NCKintJOG : NCK internal JOG active / NCK JOG interne actif
   // // MG[7].E_NCKintJOG : NCK internal JOG active / NCK JOG interne actif
   // // MG[8].E_NCKintJOG : NCK internal JOG active / NCK JOG interne actif
   // // MG[9].E_NCKintJOG : NCK internal JOG active / NCK JOG interne actif
   // // MG[10].E_NCKintJOG : NCK internal JOG active / NCK JOG interne actif
   // // MG[3].E_ChanReset : All channels in reset state / Tous les canaux en mode Reset
   // // MG[4].E_ChanReset : All channels in reset state / Tous les canaux en mode Reset
   // // MG[5].E_ChanReset : All channels in reset state / Tous les canaux en mode Reset
   // // MG[6].E_ChanReset : All channels in reset state / Tous les canaux en mode Reset
   // // MG[7].E_ChanReset : All channels in reset state / Tous les canaux en mode Reset
   // // MG[8].E_ChanReset : All channels in reset state / Tous les canaux en mode Reset
   // // MG[9].E_ChanReset : All channels in reset state / Tous les canaux en mode Reset
   // // MG[10].E_ChanReset : All channels in reset state / Tous les canaux en mode Reset
   // // MG[3].E_TEACHIN : Active machine function TEACH IN / Fonction machine active TEACH IN
   // // MG[4].E_TEACHIN : Active machine function TEACH IN / Fonction machine active TEACH IN
   // // MG[5].E_TEACHIN : Active machine function TEACH IN / Fonction machine active TEACH IN
   // // MG[6].E_TEACHIN : Active machine function TEACH IN / Fonction machine active TEACH IN
   // // MG[7].E_TEACHIN : Active machine function TEACH IN / Fonction machine active TEACH IN
   // // MG[8].E_TEACHIN : Active machine function TEACH IN / Fonction machine active TEACH IN
   // // MG[9].E_TEACHIN : Active machine function TEACH IN / Fonction machine active TEACH IN
   // // MG[10].E_TEACHIN : Active machine function TEACH IN / Fonction machine active TEACH IN
   // // MG[3].E_REPOS : Active machine function REPOS / Fonction machine active REPOS
   // // MG[4].E_REPOS : Active machine function REPOS / Fonction machine active REPOS
   // // MG[5].E_REPOS : Active machine function REPOS / Fonction machine active REPOS
   // // MG[6].E_REPOS : Active machine function REPOS / Fonction machine active REPOS
   // // MG[7].E_REPOS : Active machine function REPOS / Fonction machine active REPOS
   // // MG[8].E_REPOS : Active machine function REPOS / Fonction machine active REPOS
   // // MG[9].E_REPOS : Active machine function REPOS / Fonction machine active REPOS
   // // MG[10].E_REPOS : Active machine function REPOS / Fonction machine active REPOS
   // // MG[3].E_REF : Active machine function REF / Fonction machine active REF
   // // MG[4].E_REF : Active machine function REF / Fonction machine active REF
   // // MG[5].E_REF : Active machine function REF / Fonction machine active REF
   // // MG[6].E_REF : Active machine function REF / Fonction machine active REF
   // // MG[7].E_REF : Active machine function REF / Fonction machine active REF
   // // MG[8].E_REF : Active machine function REF / Fonction machine active REF
   // // MG[9].E_REF : Active machine function REF / Fonction machine active REF
   // // MG[10].E_REF : Active machine function REF / Fonction machine active REF
   // // MG[3].E_INC1 : INC1
   // // MG[4].E_INC1 : INC1
   // // MG[5].E_INC1 : INC1
   // // MG[6].E_INC1 : INC1
   // // MG[7].E_INC1 : INC1
   // // MG[8].E_INC1 : INC1
   // // MG[9].E_INC1 : INC1
   // // MG[10].E_INC1 : INC1
   // // MG[3].E_INC10 : INC10
   // // MG[4].E_INC10 : INC10
   // // MG[5].E_INC10 : INC10
   // // MG[6].E_INC10 : INC10
   // // MG[7].E_INC10 : INC10
   // // MG[8].E_INC10 : INC10
   // // MG[9].E_INC10 : INC10
   // // MG[10].E_INC10 : INC10
   // // MG[3].E_INC100 : INC100
   // // MG[4].E_INC100 : INC100
   // // MG[5].E_INC100 : INC100
   // // MG[6].E_INC100 : INC100
   // // MG[7].E_INC100 : INC100
   // // MG[8].E_INC100 : INC100
   // // MG[9].E_INC100 : INC100
   // // MG[10].E_INC100 : INC100
   // // MG[3].E_INC1000 : INC1000
   // // MG[4].E_INC1000 : INC1000
   // // MG[5].E_INC1000 : INC1000
   // // MG[6].E_INC1000 : INC1000
   // // MG[7].E_INC1000 : INC1000
   // // MG[8].E_INC1000 : INC1000
   // // MG[9].E_INC1000 : INC1000
   // // MG[10].E_INC1000 : INC1000
   // // MG[3].E_INC10000 : INC10000
   // // MG[4].E_INC10000 : INC10000
   // // MG[5].E_INC10000 : INC10000
   // // MG[6].E_INC10000 : INC10000
   // // MG[7].E_INC10000 : INC10000
   // // MG[8].E_INC10000 : INC10000
   // // MG[9].E_INC10000 : INC10000
   // // MG[10].E_INC10000 : INC10000
   // // MG[3].E_INCVar : INC variable / Variable INC
   // // MG[4].E_INCVar : INC variable / Variable INC
   // // MG[5].E_INCVar : INC variable / Variable INC
   // // MG[6].E_INCVar : INC variable / Variable INC
   // // MG[7].E_INCVar : INC variable / Variable INC
   // // MG[8].E_INCVar : INC variable / Variable INC
   // // MG[9].E_INCVar : INC variable / Variable INC
   // // MG[10].E_INCVar : INC variable / Variable INC
   // // MG[3].E_ContManTravelAct : Continuous manual travel active / Mode manuel continu actif
   // // MG[4].E_ContManTravelAct : Continuous manual travel active / Mode manuel continu actif
   // // MG[5].E_ContManTravelAct : Continuous manual travel active / Mode manuel continu actif
   // // MG[6].E_ContManTravelAct : Continuous manual travel active / Mode manuel continu actif
   // // MG[7].E_ContManTravelAct : Continuous manual travel active / Mode manuel continu actif
   // // MG[8].E_ContManTravelAct : Continuous manual travel active / Mode manuel continu actif
   // // MG[9].E_ContManTravelAct : Continuous manual travel active / Mode manuel continu actif
   // // MG[10].E_ContManTravelAct : Continuous manual travel active / Mode manuel continu actif
   // // MG[3].E_HMI_INC1 : INC1 from HMI / INC1 depuis IHM
   // // MG[4].E_HMI_INC1 : INC1 from HMI / INC1 depuis IHM
   // // MG[5].E_HMI_INC1 : INC1 from HMI / INC1 depuis IHM
   // // MG[6].E_HMI_INC1 : INC1 from HMI / INC1 depuis IHM
   // // MG[7].E_HMI_INC1 : INC1 from HMI / INC1 depuis IHM
   // // MG[8].E_HMI_INC1 : INC1 from HMI / INC1 depuis IHM
   // // MG[9].E_HMI_INC1 : INC1 from HMI / INC1 depuis IHM
   // // MG[10].E_HMI_INC1 : INC1 from HMI / INC1 depuis IHM
   // // MG[3].E_HMI_INC10 : INC10 from HMI / INC10 depuis IHM
   // // MG[4].E_HMI_INC10 : INC10 from HMI / INC10 depuis IHM
   // // MG[5].E_HMI_INC10 : INC10 from HMI / INC10 depuis IHM
   // // MG[6].E_HMI_INC10 : INC10 from HMI / INC10 depuis IHM
   // // MG[7].E_HMI_INC10 : INC10 from HMI / INC10 depuis IHM
   // // MG[8].E_HMI_INC10 : INC10 from HMI / INC10 depuis IHM
   // // MG[9].E_HMI_INC10 : INC10 from HMI / INC10 depuis IHM
   // // MG[10].E_HMI_INC10 : INC10 from HMI / INC10 depuis IHM
   // // MG[3].E_HMI_INC100 : INC100 from HMI / INC100 depuis IHM
   // // MG[4].E_HMI_INC100 : INC100 from HMI / INC100 depuis IHM
   // // MG[5].E_HMI_INC100 : INC100 from HMI / INC100 depuis IHM
   // // MG[6].E_HMI_INC100 : INC100 from HMI / INC100 depuis IHM
   // // MG[7].E_HMI_INC100 : INC100 from HMI / INC100 depuis IHM
   // // MG[8].E_HMI_INC100 : INC100 from HMI / INC100 depuis IHM
   // // MG[9].E_HMI_INC100 : INC100 from HMI / INC100 depuis IHM
   // // MG[10].E_HMI_INC100 : INC100 from HMI / INC100 depuis IHM
   // // MG[3].E_HMI_INC1000 : INC1000 from HMI / INC1000 depuis IHM
   // // MG[4].E_HMI_INC1000 : INC1000 from HMI / INC1000 depuis IHM
   // // MG[5].E_HMI_INC1000 : INC1000 from HMI / INC1000 depuis IHM
   // // MG[6].E_HMI_INC1000 : INC1000 from HMI / INC1000 depuis IHM
   // // MG[7].E_HMI_INC1000 : INC1000 from HMI / INC1000 depuis IHM
   // // MG[8].E_HMI_INC1000 : INC1000 from HMI / INC1000 depuis IHM
   // // MG[9].E_HMI_INC1000 : INC1000 from HMI / INC1000 depuis IHM
   // // MG[10].E_HMI_INC1000 : INC1000 from HMI / INC1000 depuis IHM
   // // MG[3].E_HMI_INC10000 : INC10000 from HMI / INC10000 depuis IHM
   // // MG[4].E_HMI_INC10000 : INC10000 from HMI / INC10000 depuis IHM
   // // MG[5].E_HMI_INC10000 : INC10000 from HMI / INC10000 depuis IHM
   // // MG[6].E_HMI_INC10000 : INC10000 from HMI / INC10000 depuis IHM
   // // MG[7].E_HMI_INC10000 : INC10000 from HMI / INC10000 depuis IHM
   // // MG[8].E_HMI_INC10000 : INC10000 from HMI / INC10000 depuis IHM
   // // MG[9].E_HMI_INC10000 : INC10000 from HMI / INC10000 depuis IHM
   // // MG[10].E_HMI_INC10000 : INC10000 from HMI / INC10000 depuis IHM
   // // MG[3].E_HMI_INCVar : INC variable from HMI / Variable INC depuis IHM
   // // MG[4].E_HMI_INCVar : INC variable from HMI / Variable INC depuis IHM
   // // MG[5].E_HMI_INCVar : INC variable from HMI / Variable INC depuis IHM
   // // MG[6].E_HMI_INCVar : INC variable from HMI / Variable INC depuis IHM
   // // MG[7].E_HMI_INCVar : INC variable from HMI / Variable INC depuis IHM
   // // MG[8].E_HMI_INCVar : INC variable from HMI / Variable INC depuis IHM
   // // MG[9].E_HMI_INCVar : INC variable from HMI / Variable INC depuis IHM
   // // MG[10].E_HMI_INCVar : INC variable from HMI / Variable INC depuis IHM
   // // MG[3].E_HMI_ContManTravel : Continuous manual travel active from HMI / Course manuelle continue active depuis IHM
   // // MG[4].E_HMI_ContManTravel : Continuous manual travel active from HMI / Course manuelle continue active depuis IHM
   // // MG[5].E_HMI_ContManTravel : Continuous manual travel active from HMI / Course manuelle continue active depuis IHM
   // // MG[6].E_HMI_ContManTravel : Continuous manual travel active from HMI / Course manuelle continue active depuis IHM
   // // MG[7].E_HMI_ContManTravel : Continuous manual travel active from HMI / Course manuelle continue active depuis IHM
   // // MG[8].E_HMI_ContManTravel : Continuous manual travel active from HMI / Course manuelle continue active depuis IHM
   // // MG[9].E_HMI_ContManTravel : Continuous manual travel active from HMI / Course manuelle continue active depuis IHM
   // // MG[10].E_HMI_ContManTravel : Continuous manual travel active from HMI / Course manuelle continue active depuis IHM
   // // MG[2] : next mode group from DBB20, as before / groupe de mode suivant depuis DBB20, comme avant
   // // MG[3] : next mode group from DBB20, as before / groupe de mode suivant depuis DBB20, comme avant
   // // MG[4] : next mode group from DBB20, as before / groupe de mode suivant depuis DBB20, comme avant
   // // MG[5] : next mode group from DBB20, as before / groupe de mode suivant depuis DBB20, comme avant
   // // MG[6] : next mode group from DBB20, as before / groupe de mode suivant depuis DBB20, comme avant
   // // MG[7] : next mode group from DBB20, as before / groupe de mode suivant depuis DBB20, comme avant
   // // MG[8] : next mode group from DBB20, as before / groupe de mode suivant depuis DBB20, comme avant
   // // MG[9] : next mode group from DBB20, as before / groupe de mode suivant depuis DBB20, comme avant
   // // MG[10] : next mode group from DBB20, as before / groupe de mode suivant depuis DBB20, comme avant
END_TYPE

